Staubli VAL3: start.pgx

program start()
begin
  //2016.07.01
  //三个任务
  //1. 运动
  //2. 获取当前位置
  //3. 人机界面


  // call View()
  //异步任务
  taskCreate "move",100,Move()
  taskCreate "View",100,View()

  taskCreateSync "postion",0.004,bOver,Postion()






end
